Xinje XDPPro project, PLC1: XL3-16 (software 3.7.17c 2024-04-02)

PROGRAM Ladder

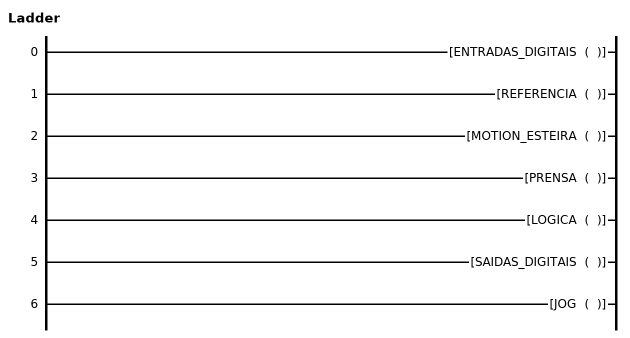
ENTRADAS_DIGITAIS ( )
REFERENCIA ( )
MOTION_ESTEIRA ( )
PRENSA ( )
LOGICA ( )
SAIDAS_DIGITAIS ( )
JOG    ( )

PROGRAM REFERENCIA

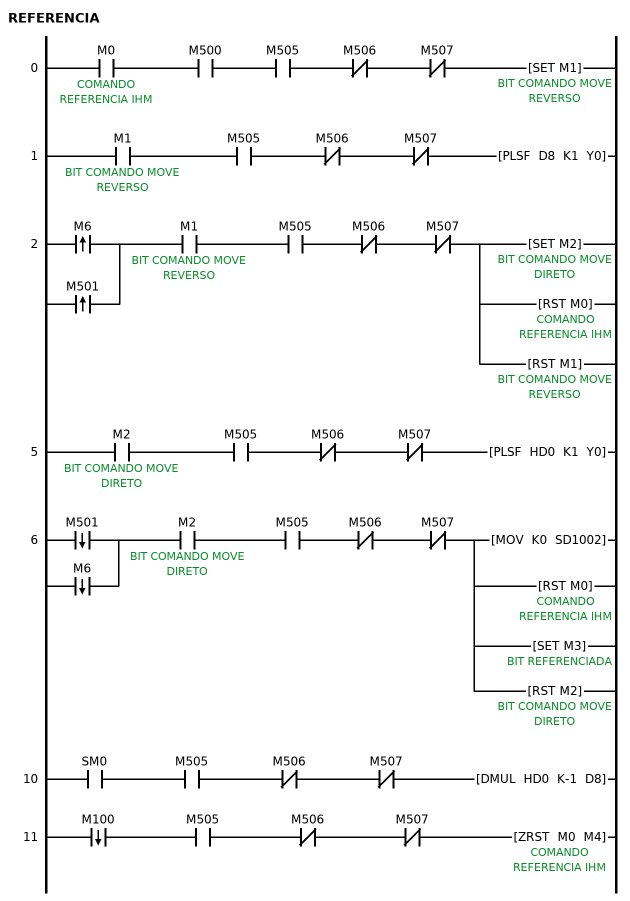
LD     M0	; COMANDO REFERENCIA IHM
AND    M500
AND    M505
ANI    M506
ANI    M507
SET    M1	; BIT COMANDO MOVE REVERSO
LD     M1	; BIT COMANDO MOVE REVERSO
AND    M505
ANI    M506
ANI    M507
PLSF   D8 K1 Y0
LDP    M6
ORP    M501
AND    M1	; BIT COMANDO MOVE REVERSO
AND    M505
ANI    M506
ANI    M507
SET    M2	; BIT COMANDO MOVE DIRETO
RST    M0	; COMANDO REFERENCIA IHM
RST    M1	; BIT COMANDO MOVE REVERSO
LD     M2	; BIT COMANDO MOVE DIRETO
AND    M505
ANI    M506
ANI    M507
PLSF   HD0 K1 Y0
LDF    M501
ORF    M6
AND    M2	; BIT COMANDO MOVE DIRETO
AND    M505
ANI    M506
ANI    M507
MOV    K0 SD1002
RST    M0	; COMANDO REFERENCIA IHM
SET    M3	; BIT REFERENCIADA
RST    M2	; BIT COMANDO MOVE DIRETO
LD     SM0
AND    M505
ANI    M506
ANI    M507
DMUL   HD0 K-1 D8
LDF    M100
AND    M505
ANI    M506
ANI    M507
ZRST   M0 M4	; COMANDO REFERENCIA IHM

PROGRAM MOTION_ESTEIRA

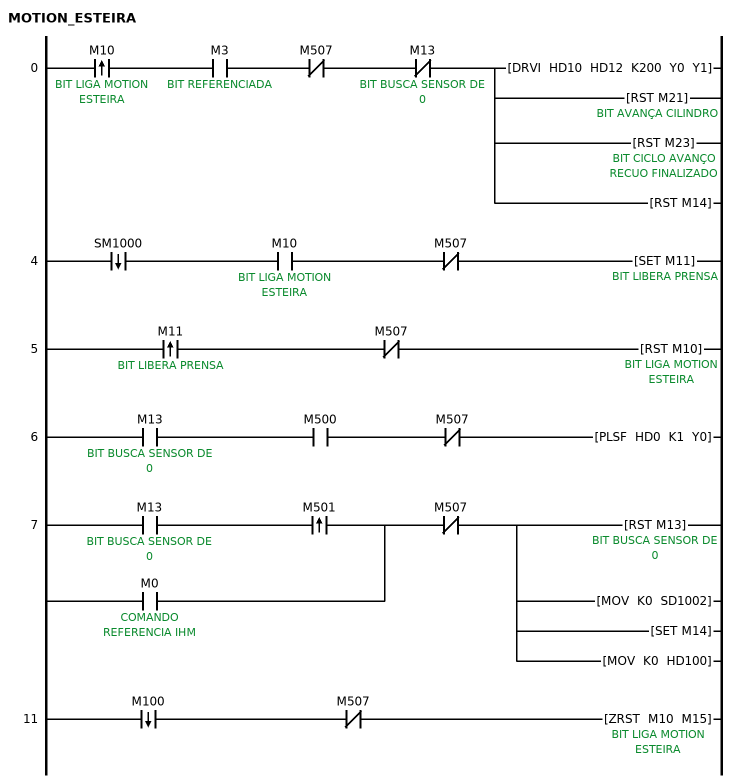
LDP    M10	; BIT LIGA MOTION ESTEIRA
AND    M3	; BIT REFERENCIADA
ANI    M507
ANI    M13	; BIT BUSCA SENSOR DE 0
DRVI   HD10 HD12 K200 Y0 Y1
RST    M21	; BIT AVANÇA CILINDRO
RST    M23	; BIT CICLO AVANÇO RECUO FINALIZADO
RST    M14
LDF    SM1000
AND    M10	; BIT LIGA MOTION ESTEIRA
ANI    M507
SET    M11	; BIT LIBERA PRENSA
LDP    M11	; BIT LIBERA PRENSA
ANI    M507
RST    M10	; BIT LIGA MOTION ESTEIRA
LD     M13	; BIT BUSCA SENSOR DE 0
AND    M500
ANI    M507
PLSF   HD0 K1 Y0
LD     M13	; BIT BUSCA SENSOR DE 0
ANDP   M501
OR     M0	; COMANDO REFERENCIA IHM
ANI    M507
RST    M13	; BIT BUSCA SENSOR DE 0
MOV    K0 SD1002
SET    M14
MOV    K0 HD100
LDF    M100
ANI    M507
ZRST   M10 M15	; BIT LIGA MOTION ESTEIRA

PROGRAM LOGICA

PROGRAM SAIDAS_DIGITAIS

PROGRAM ENTRADAS_DIGITAIS

PROGRAM PRENSA

PROGRAM JOG

COMMENTS (devices not used above)
M510	BIT AUX ENTR DIGITAL 1 SENSOR HOME
M12	BIT GIRO COMPLETO ESTEIRA
M20	BIT RECUA INICIO
M22	BIT RECUA CILINDRO